// TwinCAT 3 PLC project PLC1
// ProgramVersion: 3.1.4024.0
// libraries:
//   Tc2_EtherCAT, * (Beckhoff Automation GmbH)
//   Tc2_Standard, * (Beckhoff Automation GmbH)
//   Tc2_System, * (Beckhoff Automation GmbH)
//   Tc2_Utilities, * (Beckhoff Automation GmbH)
//   Tc3_BA2_Common, * (Beckhoff Automation GmbH)
//   Tc3_Module, * (Beckhoff Automation GmbH)
// project tree:
//   DUTs/SMPTE Timecode/ E_SMPTE_AnalogValue.TcDUT, E_SMPTE_FrameMode.TcDUT, E_SMPTE_PartOfFrame.TcDUT, E_SMPTE_TimeController_Mode.TcDUT, E_SMPTE_TimeController_Source.TcDUT, ST_SMPTE_TimeStruct.TcDUT, ST_SMPTE_TimeStructExt.TcDUT
//   DUTs/ ST_EL4732_State.TcDUT
//   FBs/ FB_SMPTE_Receiver.TcPOU, FB_SMPTE_Sender.TcPOU, FB_SMPTE_TimeController.TcPOU
//   ITFs/ I_SMPTE_TimeController.TcIO
//   POUs/ MAIN_Sender.TcPOU, MAIN_Receiver.TcPOU
//   Tasks/ PlcTaskReceiver.TcTTO, PlcTaskSender.TcTTO
// real-time tasks:
//   TASK PlcTaskReceiver: cycle T#1ms, priority 20, ADS port 350
//   TASK PlcTaskSender: cycle T#20ms, priority 1, ADS port 351
// I/O:
//   DEVICE Device 7 (EtherCAT), AmsNetId 169.254.250.244.8.1
//     Term 1 (EK1100) [EK1100 EtherCAT Coupler (2A E-Bus)]
//       Term 2 (EL4732) [EL4732 2Ch. Ana. Output +/-10V, Oversample]
//       Term 3 (EL3702) [EL3702 2Ch. Ana. Input +/-10V, DIFF, Oversample]
//       Term 4 (EL9011) [EL9011 End Terminal]
// variable links:
//   PLC1/PLC1 Instance <-> Device 7 (EtherCAT)/Term 1 (EK1100)/Term 2 (EL4732)
//     PlcTaskSender Outputs/MAIN_Sender.SMPTE_Sender.aSMPTE_out[{0..79}] <-> Ch1 Sample {0..79}/Ch1 Value  (80 links)
//   PLC1/PLC1 Instance <-> Device 7 (EtherCAT)/Term 1 (EK1100)/Term 3 (EL3702)
//     PlcTaskReceiver Inputs/MAIN_Receiver.SMPTE_Receiver.EL3702_Samples[{1..100}] <-> Ch1 Sample {0..99}/Ch1 Value  (100 links)
//   PLC1/PLC1 Instance <-> TcCOM Objects/Object1 (TcDcExternalTimeProvider)
//     PlcTaskSender Inputs/MAIN_Sender.nSysTime <-> Outputs/nSysTime

CONFIGURATION PLC1
    RESOURCE PLC ON TwinCAT3
        TASK PlcTaskReceiver(INTERVAL := T#1ms, PRIORITY := 20);
        TASK PlcTaskSender(INTERVAL := T#20ms, PRIORITY := 1);
        PROGRAM MAIN_Receiver WITH PlcTaskReceiver : MAIN_Receiver;
        PROGRAM MAIN_Sender WITH PlcTaskSender : MAIN_Sender;
    END_RESOURCE
END_CONFIGURATION

// ---- DUTs/SMPTE Timecode/E_SMPTE_AnalogValue.TcDUT
TYPE E_SMPTE_AnalogValue :
(
	LOW := 0, HIGH := 32000
)INT;
END_TYPE

// ---- DUTs/SMPTE Timecode/E_SMPTE_FrameMode.TcDUT
{attribute 'qualified_only'}
{attribute 'strict'}
TYPE E_SMPTE_FrameMode :
(
	FPS_25
);
END_TYPE

// ---- DUTs/SMPTE Timecode/E_SMPTE_PartOfFrame.TcDUT
{attribute 'qualified_only'}
{attribute 'strict'}
TYPE E_SMPTE_PartOfFrame :
(
	first := 0, second := 1
)BYTE;
END_TYPE

// ---- DUTs/SMPTE Timecode/E_SMPTE_TimeController_Mode.TcDUT
{attribute 'qualified_only'}
{attribute 'strict'}
TYPE E_SMPTE_TimeController_Mode :
(
	Stopped := 0,
	Playing := 1,
	Paused := 2
);
END_TYPE

// ---- DUTs/SMPTE Timecode/E_SMPTE_TimeController_Source.TcDUT
{attribute 'qualified_only'}
{attribute 'strict'}
TYPE E_SMPTE_TimeController_Source :
(
	NT_Time := 0,
	DC_Time := 1,
	ExtTimeProvider := 2
);
END_TYPE

// ---- DUTs/SMPTE Timecode/ST_SMPTE_TimeStruct.TcDUT
TYPE ST_SMPTE_TimeStruct :
STRUCT
	Hours: BYTE; 		// 0..24 h
	Minutes: BYTE; 		// 0..60 min
	Seconds: BYTE;		// 0..60 sec
	Frames: BYTE;		// 0..24|25|30 frames
END_STRUCT
END_TYPE

// ---- DUTs/SMPTE Timecode/ST_SMPTE_TimeStructExt.TcDUT
// Extended time struct
TYPE ST_SMPTE_TimeStructExt EXTENDS ST_SMPTE_TimeStruct :
STRUCT
	FramesUnits: BYTE;
	FramesTens: BYTE;
	SecondsUnits: BYTE;
	SecondsTens: BYTE;
	MinutesUnits: BYTE;
	MinutesTens: BYTE;
	HoursUnits: BYTE;
	HoursTens: BYTE;
END_STRUCT
END_TYPE

// ---- DUTs/ST_EL4732_State.TcDUT
TYPE ST_EL4732_State :
STRUCT
	WcState AT %I*: BYTE;
	ImfoData_State AT %I*: UINT;
	InfoData_DcOutputShift AT %I*: DINT;
	InfoData_DDcInputShift AT %I*: DINT;
END_STRUCT
END_TYPE

// ---- ITFs/I_SMPTE_TimeController.TcIO
INTERFACE I_SMPTE_TimeController

METHOD Cycle : BOOL
VAR_INPUT
END_VAR
END_METHOD

// Will pause the time
METHOD Pause : BOOL
VAR_INPUT
	bExecute : BOOL;
END_VAR
END_METHOD

PROPERTY Paused : BOOL
GET
END_GET
END_PROPERTY

// Starts the time
METHOD Play : BOOL
VAR_INPUT
	bExecute : BOOL;
END_VAR
END_METHOD

PROPERTY Playing : BOOL
GET
END_GET
END_PROPERTY

// Resets the time
METHOD Reset : BOOL
VAR_INPUT
	bExecute : BOOL;
END_VAR
END_METHOD

// Will stop the time and reset to 00:00:00:00
METHOD Stop : BOOL
VAR_INPUT
	bExecute : BOOL;
END_VAR
END_METHOD

PROPERTY Stopped : BOOL
GET
END_GET
END_PROPERTY

// Returns the SMPTE_Sender_TimeStruct
PROPERTY TimeStruct : REFERENCE TO ST_SMPTE_TimeStruct;
GET
END_GET
END_PROPERTY

END_INTERFACE

// ---- POUs/MAIN_Receiver.TcPOU
PROGRAM MAIN_Receiver
VAR
	// SMPTE Receiver
	SMPTE_Receiver 	: FB_SMPTE_Receiver;
	ReceivingSignal	: BOOL;
	FrameRate		: REAL;
	TimeString		: STRING;
	TimeStruct		: ST_SMPTE_TimeStruct;
END_VAR

(************************)
(**** SMPTE Receiver ****)
(************************)

// Call the execute method once each cycle
SMPTE_Receiver.Cycle();
// Check if the cable is connected and receiving timecode analog signal
ReceivingSignal := SMPTE_Receiver.Receiving;
// Get the framerate
FrameRate := SMPTE_Receiver.FrameRate;
// Get the time as string output
TimeString := SMPTE_Receiver.TimeString;
// Get the time as time struct
TimeStruct := SMPTE_Receiver.TimeStruct;

END_PROGRAM

// ---- FBs/FB_SMPTE_Receiver.TcPOU
FUNCTION_BLOCK FB_SMPTE_Receiver
VAR
	EL3702_Samples AT %I*: ARRAY[1..OversamplingFactor] OF INT;
	EL3702_Samples_Doublecycles : ARRAY[1..DoubleOversamplingFactor] OF INT;
	EL3702_Samples_DoublecyclesTrig : ARRAY[1..DoubleOversamplingFactor] OF INT;
	Tab_TimeCodeFrame: ARRAY[1..TimeCodeFrame] OF BYTE;					(* Bit read in the frame *)
	LastTimeCodeFrame: ARRAY[0..79] OF BYTE;									(* Last and unique TimeCode Frame *)
	SyncWord : ARRAY [1..16] OF BYTE :=[ 0, 0, 1, 1, 1, 1, 1, 1, 1, 1, 1, 1, 1, 1, 0, 1];
	SyncWordTemp : ARRAY [1..16] OF BYTE;
	i: WORD;
	j: DWORD;
	LastEdge: DWORD;
	ConstantTime: DWORD;
	Even: BOOL;	(* Is use to mesure 2 half period to detect a bit 1 *)
	First_BitZero_Reach: BOOL  := FALSE ;	(* We can mesure only when we reach a first Bit 0 otherwise we do not know in which half period of a bit 1 we are *)
	Index_Tab_EL3702: INT := 102;
	Index_Tab_TimeCodeFrame: WORD := 1;
	h: WORD;

	Index_Tab_EL3702_Error: WORD;			(* Increased when an edge had not beed detected in the last cycle *)
	Index_Tab_TimeCodeFrame_Error: WORD;	(* Increased when we are not able to catch a SyncWord in the big Array of TimeCode Bits. Normally, an Syncword each 80 bits *)
	
	// Internal Properties
	_Reset : BOOL;
	_Receiving : BOOL;
	_FrameRate: REAL;
	_FrameError: DWORD;
	
	_SMPTE_TimeStruct : ST_SMPTE_TimeStruct;
	_SMPTE_TimeStructExt : ST_SMPTE_TimeStructExt;

	_FrameRead: DWORD;
	_Time_String: STRING;
END_VAR

VAR CONSTANT
	OversamplingFactor: WORD := 100;			(* EL3702 Oversampling rate = 100 samples per cycle *)
	DoubleOversamplingFactor: WORD := 200;	(*  = OversamplingFactor x 2 *)
	TimeCodeFrame : WORD := 300;				(* bits detected in the Timecode signal *)
	SignalThreshold : INT := 25;
END_VAR

METHOD Cycle : BOOL
VAR_INST
	// Check if there is a timing error
	rtTimeError : R_TRIG;
END_VAR
// Check timing error and task time
rtTimeError(CLK := UDINT_TO_LREAL(_TaskInfo[GETCURTASKINDEXEX()].CycleTime) / 10_000 <> 1);
IF rtTimeError.Q THEN
	ADSLOGSTR( msgCtrlMask := ADSLOG_MSGTYPE_ERROR OR ADSLOG_MSGTYPE_MSGBOX, msgFmtStr := 'PLC SMPTE Receiver: Execution Time Not Valid, Please set to 1ms','');
END_IF

IF _Reset THEN
	First_BitZero_Reach := FALSE;
	Index_Tab_TimeCodeFrame := 1;
	Index_Tab_EL3702 := 102;
	Even := FALSE;
	FOR i:= 1 TO TimeCodeFrame DO
		Tab_TimeCodeFrame [ i ] := 0;
	END_FOR
	_Reset := FALSE;
END_IF

IF SignalCheck() THEN
	(* We save the last 2 cycles *)
	FOR i:=1 TO OversamplingFactor DO
		EL3702_Samples_Doublecycles [ i ] := EL3702_Samples_Doublecycles [ i+OversamplingFactor ];
	END_FOR
	FOR i:=1 TO OversamplingFactor DO
		EL3702_Samples_Doublecycles [ OversamplingFactor + i ] := EL3702_Samples [i];
	END_FOR
	
	(* Now we create an ARRAY that show the binary code *)
	ConstantTime := 0;							(* ConstantTime is the duration of a constant level of the analog signal, time between 2 edges *)
	FOR i:= 1 TO 2*OversamplingFactor DO
		  EL3702_Samples_DoublecyclesTrig [i ] := 0;	(* An array that provide only the edges of the analog signal, only in the last cycle *)
	END_FOR
	
	FOR i:= Index_Tab_EL3702 TO ( 2*OversamplingFactor-1)  DO
		IF 	EL3702_Samples_Doublecycles[ i-1] * EL3702_Samples_Doublecycles [ i ] < 0					(* The analog signal change of sign --> there is an edge *)
		OR 	EL3702_Samples_Doublecycles [ i-1 ] <> 0 AND EL3702_Samples_Doublecycles [ i ] = 0 THEN	(* We capture a sample that is 0 : It's also a new edge *)
			EL3702_Samples_DoublecyclesTrig [ i ] := 1;
			IF LastEdge = 0 THEN										(* We have to wait a least the second edge to mesure *)
				LastEdge := i;
			ELSE													(* Let's go ... *)
				ConstantTime := (i - LastEdge) * 10 ;  	(* if  EL3702 Oversampling time = 10 µs*)
				LastEdge := i;
				IF ConstantTime < 330 AND ConstantTime<>0 AND First_BitZero_Reach THEN		(* It's part of a 1 signal *)
					(* 330µs is a fix limit that match all frame rates : Minimum period is 400 µs at 30 fr/sec, maximum half period is 260 µs at 24 fr/sec*)
					IF First_BitZero_Reach THEN											(* We first need to read a 0 bit, or we are not able to know in wich part of a 1 bit we are *)
						IF NOT Even THEN				(* First part of a 1 bit *)
							Index_Tab_EL3702 := i ;
							Even := TRUE;
						ELSE							(* Second part of a 1 bit *)
							Tab_TimeCodeFrame [ Index_Tab_TimeCodeFrame ] := 1;			(* We save a 1 bit in an array *)
							Index_Tab_TimeCodeFrame := Index_Tab_TimeCodeFrame + 1;		(* and manage this array *)
							Index_Tab_EL3702 := i ;										(* This bit in Frame is already handled, we will continu from this sample *)
							Even := FALSE;
						END_IF
					END_IF
				ELSIF ConstantTime > 300  THEN											(* It's a 0 bit *)
					First_BitZero_Reach := TRUE; 											(* One 0 bit had been detected. We are now able to mesure 1 bit *)
					IF Even THEN						(* If we were in the first part of a 1 bit *)
						Even := FALSE;
						_FrameError := _FrameError + 1;		(* Then this 1 bit is not finished and it's a Frame Error *)
					END_IF
					Tab_TimeCodeFrame [ Index_Tab_TimeCodeFrame ] := 0;					(* We save a 1 bit in an array *)
					Index_Tab_TimeCodeFrame := Index_Tab_TimeCodeFrame + 1;				(* and manage this array *)
					Index_Tab_EL3702 := i ;												(* This bit in Frame is already handled, we will continu from this sample *)
					_FrameRate := 1000000.0 / (ConstantTime * 80);	(* We measure the frame Rate. 0 Signal = 1 bit. 80 bit / frame *)
				END_IF
			END_IF
		END_IF
	END_FOR
	Index_Tab_EL3702 := Index_Tab_EL3702 - OversamplingFactor +1; 			(* +1 in order to do not take in consideration the last one we handled *)
	IF Index_Tab_EL3702 < 2  THEN							(* There is a problem : We should be able to read an edge in the last cycle *)
		Index_Tab_EL3702_Error := Index_Tab_EL3702_Error + 1;
	END_IF
	LastEdge := LastEdge - OversamplingFactor;										(* We will shift the array of the last 2 Oversampling cycle. Then the last Edge will be 100 samples before *)
	
	
	
	
	(* We are looking for the SyncWord - Sequence 0, 0, 1, 1, 1, 1, 1, 1, 1, 1, 1, 1, 1, 1, 0, 1 *)
	FOR i:=16 TO  ( TimeCodeFrame ) DO	(* Sync Word = 16 bits *)
		FOR j := 1 TO 16 DO
			SyncWordTemp [ j ] := Tab_TimeCodeFrame [ i -16 + j ]; 				(* Part of the Array that contain all bits read from the Timecode Frame *)
		END_FOR
		IF MEMCMP( ADR(SyncWord) , ADR(SyncWordTemp), 16) = 0 THEN		(* We compare this part with the SynWord *)
			IF i >= 80 THEN	(* A SyncWord is found and all bits that are in this frame are available *)
					MEMCPY( ADR(LastTimeCodeFrame) , ADR(Tab_TimeCodeFrame) + i  - 80, 80);	(* We extract this TimeCode Frame from the complete array *)
					
					_SMPTE_TimeStructExt.FramesUnits := LastTimeCodeFrame [0] * 1
													+LastTimeCodeFrame [1] * 2
													+LastTimeCodeFrame [2] * 4
													+LastTimeCodeFrame [3] * 8;
													
					_SMPTE_TimeStructExt.FramesTens :=  LastTimeCodeFrame [8] * 10
													+LastTimeCodeFrame [9] * 20;
													
					_SMPTE_TimeStructExt.SecondsUnits := LastTimeCodeFrame [16] * 1
													 +LastTimeCodeFrame [17] * 2
													 +LastTimeCodeFrame [18] * 4
													 +LastTimeCodeFrame [19] * 8;
													 
					_SMPTE_TimeStructExt.SecondsTens := LastTimeCodeFrame [24] * 10
													+LastTimeCodeFrame [25] * 20
													+LastTimeCodeFrame [26] * 40;
													
					_SMPTE_TimeStructExt.MinutesUnits := LastTimeCodeFrame [32] * 1
													 +LastTimeCodeFrame [33] * 2
													 +LastTimeCodeFrame [34] * 4
													 +LastTimeCodeFrame [35] * 8;
													 
					_SMPTE_TimeStructExt.MinutesTens := LastTimeCodeFrame [40] * 10
													+LastTimeCodeFrame [41] * 20
													+LastTimeCodeFrame [42] * 40;
													
					_SMPTE_TimeStructExt.HoursUnits := LastTimeCodeFrame [48] * 1
												   +LastTimeCodeFrame [49] * 2
												   +LastTimeCodeFrame [50] * 4
												   +LastTimeCodeFrame [51] * 8;
												   
					_SMPTE_TimeStructExt.HoursTens := LastTimeCodeFrame [56] * 10
												   +LastTimeCodeFrame [57] * 20;
												   

					_SMPTE_TimeStructExt.Frames := _SMPTE_TimeStructExt.FramesTens + _SMPTE_TimeStructExt.FramesUnits;
					_SMPTE_TimeStructExt.Seconds := _SMPTE_TimeStructExt.SecondsTens + _SMPTE_TimeStructExt.SecondsUnits;
					_SMPTE_TimeStructExt.Minutes := _SMPTE_TimeStructExt.MinutesTens + _SMPTE_TimeStructExt.MinutesUnits;
					_SMPTE_TimeStructExt.Hours := _SMPTE_TimeStructExt.HoursTens + _SMPTE_TimeStructExt.HoursUnits;
					
					_SMPTE_TimeStruct.Frames  := _SMPTE_TimeStructExt.Frames;
					_SMPTE_TimeStruct.Seconds := _SMPTE_TimeStructExt.Seconds;
					_SMPTE_TimeStruct.Minutes := _SMPTE_TimeStructExt.Minutes;
					_SMPTE_TimeStruct.Hours   := _SMPTE_TimeStructExt.Hours;
					
					_Time_String := CONCAT ( INT_TO_STRING (_SMPTE_TimeStructExt.Hours), ' : ');
					_Time_String := CONCAT (_Time_String,  INT_TO_STRING (_SMPTE_TimeStructExt.Minutes));
					_Time_String := CONCAT (_Time_String,  ' : ');
					_Time_String := CONCAT (_Time_String,  INT_TO_STRING (_SMPTE_TimeStructExt.Seconds));
					_Time_String := CONCAT (_Time_String,  ' : ');
					_Time_String := CONCAT (_Time_String,  INT_TO_STRING (_SMPTE_TimeStructExt.Frames));
	
					_FrameRead := _FrameRead + 1; 							(* Number of frame read *)
	
					FOR h:=1 TO (TimeCodeFrame - i ) DO							(* Now, we suppress this TimeCode frame from the array of bit, and shift this array *)
						Tab_TimeCodeFrame [ h ] := Tab_TimeCodeFrame [ h + i ];
					END_FOR
					FOR h:= (TimeCodeFrame - i ) TO TimeCodeFrame DO
						Tab_TimeCodeFrame [ h ] := 0;
					END_FOR
	
					 Index_Tab_TimeCodeFrame := Index_Tab_TimeCodeFrame - i ;		(* Next bit in the frame will be place here now *)
	
					EXIT ;
			END_IF
		END_IF
	END_FOR
	
	IF Index_Tab_TimeCodeFrame > TimeCodeFrame THEN	(* There is a problem : We should be able to catch a SyncWord in a so big array a Timecode bit. Normally a SyncWord each 80 bits*)
		Index_Tab_TimeCodeFrame_Error := Index_Tab_TimeCodeFrame_Error + 1;
		Reset := TRUE;
	END_IF
END_IF
END_METHOD

PROPERTY FrameError : DWORD
GET
FrameError := _FrameError;
END_GET
END_PROPERTY

PROPERTY FrameRate : REAL
GET
FrameRate := _FrameRate;
END_GET
END_PROPERTY

PROPERTY FramesReceived : DWORD
GET
FramesReceived := _FrameRead;
END_GET
END_PROPERTY

PROPERTY Receiving : BOOL
GET
Receiving := _Receiving;
END_GET
END_PROPERTY

PROPERTY Reset : BOOL
SET
_Reset := Reset;
END_SET
END_PROPERTY

METHOD INTERNAL SignalCheck : BOOL
VAR
	itr_X : INT;
END_VAR
// Check for EL3702 is receiving signals, plugged into device
_Receiving := FALSE;
FOR itr_X := 1 TO 100 DO
	IF EL3702_Samples[itr_X] >= SignalThreshold OR EL3702_Samples[itr_X] <= (SignalThreshold * -1) THEN
		SignalCheck := TRUE;
		_Receiving := TRUE;
		EXIT;
	END_IF
END_FOR
END_METHOD

PROPERTY TimeString : REFERENCE TO STRING
GET
TimeString REF= _Time_String;
END_GET
END_PROPERTY

PROPERTY TimeStruct : REFERENCE TO ST_SMPTE_TimeStruct
GET
TimeStruct REF= _SMPTE_TimeStruct;
END_GET
END_PROPERTY

PROPERTY TimeStructExt : REFERENCE TO ST_SMPTE_TimeStructExt
GET
TimeStructExt REF= _SMPTE_TimeStructExt;
END_GET
END_PROPERTY

END_FUNCTION_BLOCK

// ---- POUs/MAIN_Sender.TcPOU
PROGRAM MAIN_Sender
VAR
	// SMPTE Time Controller
	SMPTE_TimeController : FB_SMPTE_TimeController(eTimeSource := E_SMPTE_TimeController_Source.ExtTimeProvider, eFrameMode := E_SMPTE_FrameMode.FPS_25);
	// SMPTE Sender
	SMPTE_Sender 	: FB_SMPTE_Sender(ipSMPTE_TimeController := SMPTE_TimeController);
	
	// External Time Source
	nSysTime AT %I* : ULINT;
	
	// Enable the sender
	bEnableSending: BOOL;
	// Disable the sender
	bDisableSending: BOOL;
	// Error status of sender
	bSMPTE_Error: BOOL;
	// Enable Status
	bSMPTE_Enabled: BOOL;
	
	// Play the timeline
	bPlay: BOOL;
	// Pause the timeline
	bPause: BOOL;
	// Stop the timeline
	bStop: BOOL;
	// Reset the timeline
	bReset: BOOL;
	
	// View the current time struct being send
	stSMPTE_TimeStruct : ST_SMPTE_TimeStruct;

END_VAR

(**********************)
(**** SMPTE Sender ****)
(**********************)

// Call once each cycle
SMPTE_TimeController.Cycle();
SMPTE_Sender.Cycle();

// Enable sending the SMPTE signal
IF SMPTE_Sender.EnableSending(bExecute := bEnableSending) THEN
	bEnableSending := FALSE;
END_IF

// Disable sending the SMPTE signal
IF SMPTE_Sender.DisableSending(bExecute := bDisableSending) THEN
	bDisableSending := FALSE;
END_IF

// Check if errors on SMPTE Sender
bSMPTE_Error := SMPTE_Sender.Error;
// Check if enabled
bSMPTE_Enabled := SMPTE_Sender.Enabled;



(********************************)
(**** SMPTE Time Conectoller ****)
(********************************)

// Assign External Time Source
SMPTE_TimeController.AssignExternalTimeSource(nSysTime);

// Playback controls
IF SMPTE_TimeController.Play(bExecute := bPlay) THEN
	bPlay := FALSE;
END_IF

IF SMPTE_TimeController.Pause(bExecute := bPause) THEN
	bPause := FALSE;
END_IF

IF SMPTE_TimeController.Stop(bExecute := bStop) THEN
	bStop := FALSE;
END_IF

IF SMPTE_TimeController.Reset(bExecute := bReset) THEN
	bReset := FALSE;
END_IF

// Sample of Timecode being send
stSMPTE_TimeStruct := SMPTE_TimeController.TimeStruct;

END_PROGRAM

// ---- FBs/FB_SMPTE_TimeController.TcPOU
FUNCTION_BLOCK FB_SMPTE_TimeController IMPLEMENTS I_SMPTE_TimeController
VAR
	// Internal Time Source mode
	_eTimeSource : E_SMPTE_TimeController_Source;
	
	// Linked to TcCom Object for Time Provider if using Ext Mode
	_TcExternalTimeSource : REFERENCE TO ULINT; 
	
	// Frame Mode
	_eFrameMode: E_SMPTE_FrameMode := E_SMPTE_FrameMode.FPS_25;	// transmitting with 25 fps (frames per second)		
	
	// Used for DC Time
	_dcTime	: T_DCTIME64;
			
	// SMPTE Time Struct
	_stSMPTE_TimeStruct : ST_SMPTE_TimeStruct;
	
	// Reference time timestamp
	_bRefTimeInit : BOOL;
	
	// Current Time Strunct
	_CurrentTime :	TIMESTRUCT;
		
	// Current Time Value
	_RefTime : T_DCTIME64;
	
	// Working Time Value
	_WorkTime : T_DCTIME64;
	
	// Paused Time Value
	_PauseTime : T_DCTIME64;
	
	// Mode Status
	_eSMPTE_TimeController_Mode : E_SMPTE_TimeController_Mode;
	
	// Playing Status Variables
	_Playing : BOOL;
	
	// Paused Status Variables
	_Paused : BOOL;
	
	// Stopped Status Variables
	_Stopped : BOOL;
	
	// Reset Control Variables
	_Reset : BOOL;
	
	// Error, usually due to timesource
	_Error : BOOL;
END_VAR

METHOD AssignExternalTimeSource : BOOL
VAR_INPUT
	// Linked to TcCom Object for Time Provider if using Ext Mode
	TcExternalTimeSource : REFERENCE TO ULINT; 
END_VAR
_TcExternalTimeSource REF= TcExternalTimeSource;
AssignExternalTimeSource := TRUE;
END_METHOD

METHOD Cycle : BOOL
VAR_INST
	_CalcTimeDiff : FB_EcExtSyncCalcTimeDiff64;
	_bWasPaused : BOOL;
END_VAR
// Check Mode and compute time
CASE _eSMPTE_TimeController_Mode OF
	E_SMPTE_TimeController_Mode.Playing:
	
		// Get the working time
		UpdateTime(_WorkTime); 
		
		// Get the reference clock
		IF NOT _bRefTimeInit THEN
			_RefTime := _WorkTime;
			_bRefTimeInit := TRUE;
		END_IF
		
		// Recovery from Pause
		IF _bWasPaused THEN
			_RefTime := _WorkTime - _PauseTime;
			_bWasPaused := FALSE;
		END_IF

	E_SMPTE_TimeController_Mode.Paused:
		IF NOT _bWasPaused THEN
			_PauseTime := _WorkTime - _RefTime;
			_bWasPaused := TRUE;
		END_IF
	
	E_SMPTE_TimeController_Mode.Stopped:
		// Stop the clock and reset
		_bRefTimeInit := FALSE;
		_bWasPaused := FALSE;
		_PauseTime := 0;
		_WorkTime := 0;
		_RefTime := 0;
END_CASE

// If not paused, update the time stuct
IF NOT (_eSMPTE_TimeController_Mode = E_SMPTE_TimeController_Mode.Paused) THEN
	// Convert to time struct
	_CurrentTime := DCTIME64_TO_SYSTEMTIME(_WorkTime - _RefTime);
END_IF

// Reset
IF _Reset THEN
	_bRefTimeInit := FALSE;
	_bWasPaused := FALSE;
	_PauseTime := 0;
	_WorkTime := 0;
	_RefTime := 0;
	_Reset := FALSE;
END_IF

// Remove unused values
_CurrentTime.wDay := 0;
_CurrentTime.wDayOfWeek := 0;
_CurrentTime.wMonth := 0;
_CurrentTime.wYear := 0;
END_METHOD

PROPERTY Error : BOOL
GET
Error := _Error;
END_GET
END_PROPERTY

METHOD FB_init : BOOL
VAR_INPUT
	(* if TRUE, the retain variables are initialized (warm start / cold start)*)
	bInitRetains	: BOOL;
	(* if TRUE, the instance afterwards gets moved into the copy code (online change)*)
	bInCopyCode	: BOOL;
	(* Time Source*)
	eTimeSource	: E_SMPTE_TimeController_Source;
	(* Frame Mode, transmitting with 25 fps (frames per second) *)
	eFrameMode : E_SMPTE_FrameMode := E_SMPTE_FrameMode.FPS_25;
END_VAR
_eTimeSource := eTimeSource;
_eFrameMode := eFrameMode;
END_METHOD

(* Will pause the time*)
METHOD Pause : BOOL
VAR_INPUT
	bExecute	: BOOL;
END_VAR
VAR_INST
	rtExecute : R_TRIG;
END_VAR
rtExecute(CLK := bExecute);
IF rtExecute.Q THEN
	_eSMPTE_TimeController_Mode := E_SMPTE_TimeController_Mode.Paused;
	// Return TRUE
	Pause := TRUE;
END_IF
END_METHOD

PROPERTY Paused : BOOL
GET
Paused := _eSMPTE_TimeController_Mode = E_SMPTE_TimeController_Mode.Paused;
END_GET
END_PROPERTY

(* Starts the time*)
METHOD Play : BOOL
VAR_INPUT
	bExecute	: BOOL;
END_VAR
VAR_INST
	rtExecute :  R_TRIG;
END_VAR
rtExecute(CLK := bExecute);
IF rtExecute.Q THEN
	_eSMPTE_TimeController_Mode := E_SMPTE_TimeController_Mode.Playing;
	// Return TRUE
	Play := TRUE;
END_IF
END_METHOD

PROPERTY Playing : BOOL
GET
Playing := _eSMPTE_TimeController_Mode = E_SMPTE_TimeController_Mode.Playing;
END_GET
END_PROPERTY

(* Resets the time*)
METHOD Reset : BOOL
VAR_INPUT
	bExecute	: BOOL;
END_VAR
VAR_INST
	rtExecute :  R_TRIG;
END_VAR
rtExecute(CLK := bExecute);
IF rtExecute.Q THEN
	_Reset := TRUE;
	// Return TRUE
	Reset := TRUE;
END_IF
END_METHOD

(* Will stop the time and reset to 00:00:00:00*)
METHOD Stop : BOOL
VAR_INPUT
	bExecute	: BOOL;
END_VAR
VAR_INST
	rtExecute :  R_TRIG;
END_VAR
rtExecute(CLK := bExecute);
IF rtExecute.Q THEN
	_eSMPTE_TimeController_Mode := E_SMPTE_TimeController_Mode.Stopped;
	// Return TRUE
	Stop := TRUE;
END_IF
END_METHOD

PROPERTY Stopped : BOOL
GET
Stopped := _eSMPTE_TimeController_Mode = E_SMPTE_TimeController_Mode.Stopped;
END_GET
END_PROPERTY

(* Returns the SMPTE_TimeStruct*)
PROPERTY TimeStruct : REFERENCE TO ST_SMPTE_TimeStruct;
GET
// Compute the Time Struct for SMPTE
CASE _eFrameMode OF
	E_SMPTE_FrameMode.FPS_25:
		_stSMPTE_TimeStruct.Hours := WORD_TO_BYTE(_CurrentTime.wHour);
		_stSMPTE_TimeStruct.Minutes := WORD_TO_BYTE(_CurrentTime.wMinute);
		_stSMPTE_TimeStruct.Seconds := WORD_TO_BYTE(_CurrentTime.wSecond);
		_stSMPTE_TimeStruct.Frames := DINT_TO_BYTE(TRUNC(WORD_TO_REAL(_CurrentTime.wMilliseconds)/(1000/25)));
END_CASE

// Return the time struct
TimeStruct REF= _stSMPTE_TimeStruct;
END_GET
END_PROPERTY

METHOD INTERNAL UpdateTime: BOOL;
VAR_IN_OUT
	// Current Time Struct
	_CurDCTime : T_DCTIME64;
END_VAR
VAR_INST
	// Used for NT Time
	_ntTime	: TIMESTRUCT;
	_ntGetTime : NT_GetTime;
	// Ref Error Trig
	rtRefError : R_TRIG; 
END_VAR
// Check for reference error on External time source
rtRefError(CLK := NOT __ISVALIDREF(_TcExternalTimeSource));
IF rtRefError.Q THEN
	ADSLOGSTR( msgCtrlMask := ADSLOG_MSGTYPE_ERROR OR ADSLOG_MSGTYPE_MSGBOX, msgFmtStr := 'PLC SMPTE Time Controller: Invalid Timesource Provided or Disconnected: Use AssignExternalTimeSource()','');
END_IF

// Calculate the time
CASE _eTimeSource OF
	E_SMPTE_TimeController_Source.ExtTimeProvider:
		(* External Time Provider *)
		IF __ISVALIDREF(_TcExternalTimeSource) THEN
			_dcTime := FILETIME64_TO_DCTIME64(_TcExternalTimeSource);
			_CurDCTime := _dcTime;
			_Error := FALSE;
		ELSE
			_eSMPTE_TimeController_Mode := E_SMPTE_TimeController_Mode.Stopped;
			_Error := TRUE;
		END_IF
	
	E_SMPTE_TimeController_Source.DC_Time:
		(* External Time Provider *)
		_dcTime := F_GetCurDcTickTime64();
		_CurDCTime := _dcTime;
	
	E_SMPTE_TimeController_Source.NT_Time:
		(* NT Time Provider *)
		IF NOT _ntGetTime.BUSY THEN
			_ntGetTime(start := TRUE, TIMESTR => _ntTime);
		END_IF
		_ntGetTime(start := FALSE);
		_CurDCTime := SYSTEMTIME_TO_DCTIME64(_ntTime, 0, 0);
END_CASE

UpdateTime := TRUE;
END_METHOD

END_FUNCTION_BLOCK

// ---- FBs/FB_SMPTE_Sender.TcPOU
FUNCTION_BLOCK FB_SMPTE_Sender
VAR
	// Analog Signal Output
	aSMPTE_out AT%Q*: ARRAY[0..79] OF E_SMPTE_AnalogValue;
	
	// Status Variables
	_bEnabled: BOOL; // Enabled
	_bError: BOOL;	// becomes true, if plc cycle time <> 20ms	
	_bReady: BOOL;	// two cycles are needed to transmitt a comlete message - the FB accepts data only if READY!
	
	// SMPTE Time Contrller Object
	_ipSMPTE_TimeController : I_SMPTE_TimeController;
		
	// Internal Variables
	eCurrentPart: E_SMPTE_PartOfFrame := E_SMPTE_PartOfFrame.first;
	nPos: BYTE;
	aTmp: ARRAY[0..3] OF BOOL;

	// Internal Time Struct
	_stSMPTE_TimeStruct: ST_SMPTE_TimeStruct;
END_VAR

METHOD INTERNAL ChangePart  : HResult
VAR_IN_OUT
	eCurrentPartOfFrame : E_SMPTE_PartOfFrame;
END_VAR
eCurrentPartOfFrame := sel(eCurrentPartOfFrame = E_SMPTE_PartOfFrame.first, E_SMPTE_PartOfFrame.first, E_SMPTE_PartOfFrame.second);
END_METHOD

METHOD Cycle : BOOL
VAR_INST
	rTrigEnable: R_TRIG;
	fTrigEnable: F_TRIG;
	// Check if there is a timing error
	rtTimeError : R_TRIG;
END_VAR
// Check timing error and task time
rtTimeError(CLK := UDINT_TO_LREAL(_TaskInfo[GETCURTASKINDEXEX()].CycleTime) / 10_000 <> 20);
IF rtTimeError.Q THEN
	ADSLOGSTR( msgCtrlMask := ADSLOG_MSGTYPE_ERROR OR ADSLOG_MSGTYPE_MSGBOX, msgFmtStr := 'PLC SMPTE Sender: Execution Time Not Valid, Please set to 20ms','');
END_IF

rTrigEnable(CLK := _bEnabled);
fTrigEnable(CLK := _bEnabled);

IF fTrigEnable.Q THEN
	_bReady := FALSE;
ELSIF rTrigEnable.Q THEN
	eCurrentPart := E_SMPTE_PartOfFrame.first;
	// cycle time using this FB must be 20ms - reason: Oversampling terminal!
	_bError := UDINT_TO_LREAL(_TaskInfo[GETCURTASKINDEXEX()].CycleTime) / 10_000 <> 20;
END_IF	

// Check if time source is valid and configured
IF (_ipSMPTE_TimeController = 0) THEN
	_bError := TRUE;
END_IF

// Check if there are errors or if no enabled
IF NOT _bEnabled OR _bError THEN
	RETURN;
END_IF
	
nPos := 0;
IF eCurrentPart = E_SMPTE_PartOfFrame.first THEN
	_stSMPTE_TimeStruct := _ipSMPTE_TimeController.TimeStruct;	// accept input value now!
	{region 'Frames (including userbits)'}
	Write_4Bits(aSMPTE_out,nPos, GetBits(_stSMPTE_TimeStruct.Frames, FALSE));
	Write_4Bits(aSMPTE_out,nPos, GetBits(0, TRUE));          
	Write_4Bits(aSMPTE_out,nPos, GetBits(_stSMPTE_TimeStruct.Frames,TRUE));
	Write_4Bits(aSMPTE_out,nPos, GetBits(0, TRUE));          
	{endregion}                                              
                                                             
	{region 'Seconds (including userbits'}                   
	Write_4Bits(aSMPTE_out,nPos, GetBits(_stSMPTE_TimeStruct.Seconds, FALSE));
	Write_4Bits(aSMPTE_out,nPos, GetBits(0, TRUE));          
	Write_4Bits(aSMPTE_out,nPos, GetBits(_stSMPTE_TimeStruct.Seconds,TRUE));
	Write_4Bits(aSMPTE_out,nPos, GetBits(0, TRUE));          
	{endregion}                                              
                                                             
	{region 'Minutes - Units only!'}                         
	Write_4Bits(aSMPTE_out,nPos, GetBits(_stSMPTE_TimeStruct.Minutes, FALSE));
	Write_4Bits(aSMPTE_out,nPos, GetBits(0, TRUE));          
	{endregion}                                              
                                                             
	_bReady := FALSE; 	                                     
		                                                     
ELSE // second part of the complete SMPTE Frame              
	{region 'Minutes - Tens only!'}                          
	Write_4Bits(aSMPTE_out,nPos, GetBits(_stSMPTE_TimeStruct.Minutes, TRUE));
	Write_4Bits(aSMPTE_out,nPos, GetBits(0, TRUE));          
	{endregion}                                              
                                                             
	{region 'hours (including userbits'}                     
	Write_4Bits(aSMPTE_out,nPos, GetBits(_stSMPTE_TimeStruct.Hours, FALSE));
	Write_4Bits(aSMPTE_out,nPos, GetBits(0, TRUE));          
	Write_4Bits(aSMPTE_out,nPos, GetBits(_stSMPTE_TimeStruct.Hours,TRUE));
	Write_4Bits(aSMPTE_out,nPos, GetBits(0, TRUE));
	{endregion}

	{region 'Syncword'}
	WriteSyncWord(aSMPTE_out,nPos);
	{endregion}
		 
	_bReady := TRUE;			 
END_IF

// one complete SMPTE frame always consists of two parts (2*20ms):
ChangePart(eCurrentPartOfFrame := eCurrentPart);
END_METHOD

METHOD DisableSending : BOOL
VAR_INPUT
	bExecute	: BOOL;
END_VAR
VAR_INST
	rtExecute : R_TRIG;
END_VAR
rtExecute(CLK := bExecute);
IF rtExecute.Q THEN
	_bEnabled := FALSE;
	// Return TRUE
	DisableSending := TRUE;
END_IF
END_METHOD

PROPERTY Enabled : BOOL
GET
Enabled := _bEnabled;
END_GET
END_PROPERTY

METHOD EnableSending : BOOL
VAR_INPUT
	bExecute	: BOOL;
END_VAR
VAR_INST
	rtExecute : R_TRIG;
END_VAR
rtExecute(CLK := bExecute);
IF rtExecute.Q THEN
	_bEnabled := TRUE;
	// Return TRUE
	EnableSending := TRUE;
END_IF
END_METHOD

PROPERTY Error : BOOL
GET
END_GET
END_PROPERTY

METHOD FB_init : BOOL
VAR_INPUT
	bInitRetains : BOOL; // if TRUE, the retain variables are initialized (warm start / cold start)
	bInCopyCode : BOOL;  // if TRUE, the instance afterwards gets moved into the copy code (online change)
	ipSMPTE_TimeController : I_SMPTE_TimeController;
END_VAR
_ipSMPTE_TimeController := ipSMPTE_TimeController;
END_METHOD

METHOD INTERNAL GetBits : ARRAY[0..3] OF BOOL
VAR_INPUT
	nValue: BYTE;
	bGetTens: BOOL;
END_VAR
VAR
	i: SINT;
END_VAR
FOR i:= 3 TO 0 BY -1 DO
	GetBits[i] := nValue >= 10* EXPT(2,i);
	nValue := LREAL_TO_BYTE(SEL(GetBits[i], nValue, nValue - (10* EXPT(2,i))));
END_FOR

IF bGetTens THEN
	RETURN;
END_IF

FOR i:= 3 TO 0 BY -1 DO
	GetBits[i] := nValue >= EXPT(2,i);
	nValue := LREAL_TO_BYTE(SEL(GetBits[i], nValue, nValue - EXPT(2,i)));
END_FOR
END_METHOD

PROPERTY Ready : BOOL
GET
END_GET
END_PROPERTY

METHOD INTERNAL Write_4Bits : HResult
VAR_IN_OUT
	aDataOut: ARRAY[0..79] OF E_SMPTE_AnalogValue;
	nPos: BYTE;
END_VAR

VAR_input
	aValue: ARRAY[0..3] OF BOOL;
END_VAR

VAR
	ePreviousAnalogValue: E_SMPTE_AnalogValue;
	i: SINT;
END_VAR
IF nPos = 0 THEN
	ePreviousAnalogValue := aDataOut[79];
	Write_4Bits := 1;
ELSE
	ePreviousAnalogValue := aDataOut[nPos-1];
	Write_4Bits := S_OK;
END_IF

FOR i:= 0 TO 3 DO
	IF aValue[i] THEN
		IF ePreviousAnalogValue = E_SMPTE_AnalogValue.HIGH THEN
			aDataOut[nPos] := E_SMPTE_AnalogValue.LOW;
			aDataOut[nPos + 1] := E_SMPTE_AnalogValue.HIGH;
		ELSE
			aDataOut[nPos] := E_SMPTE_AnalogValue.HIGH;
			aDataOut[nPos + 1] := E_SMPTE_AnalogValue.LOW;
		END_IF
	ELSE
		IF ePreviousAnalogValue = E_SMPTE_AnalogValue.HIGH THEN
			aDataOut[nPos] := aDataOut[nPos + 1] := E_SMPTE_AnalogValue.LOW;
		ELSE
			aDataOut[nPos] := aDataOut[nPos + 1] := E_SMPTE_AnalogValue.HIGH;
		END_IF
	END_IF
	ePreviousAnalogValue := aDataOut[nPos + 1];
	nPos := nPos + 2;
END_FOR
END_METHOD

METHOD INTERNAL WriteSyncword: HRESULT
VAR_IN_OUT
	aDataOut: ARRAY[0..79] OF E_SMPTE_AnalogValue;
	nPos: BYTE;
END_VAR

VAR
	i: INT;
END_VAR
// Syncword: 0011.1111.1111.1101

WriteSyncword	:= S_OK;
IF nPos <> 48 THEN
	WriteSyncword	:= -3;
	RETURN;
ELSIF aDataOut[47]=  E_SMPTE_AnalogValue.HIGH THEN // create syncword based on the last analog value ...
	// 0011
	aDataOut[nPos] := E_SMPTE_AnalogValue.LOW; 		nPos := nPos + 1;
	aDataOut[nPos] := E_SMPTE_AnalogValue.LOW; 		nPos := nPos + 1;
	aDataOut[nPos] := E_SMPTE_AnalogValue.HIGH; 		nPos := nPos + 1;
	aDataOut[nPos] := E_SMPTE_AnalogValue.HIGH; 		nPos := nPos + 1;
	aDataOut[nPos] := E_SMPTE_AnalogValue.LOW; 		nPos := nPos + 1;
	aDataOut[nPos] := E_SMPTE_AnalogValue.HIGH; 		nPos := nPos + 1;
	aDataOut[nPos] := E_SMPTE_AnalogValue.LOW; 		nPos := nPos + 1;
	aDataOut[nPos] := E_SMPTE_AnalogValue.HIGH; 		nPos := nPos + 1;
	
	// 2* 1111
	FOR i:= 0 TO 1 DO 
		aDataOut[nPos] := E_SMPTE_AnalogValue.LOW; 		nPos := nPos + 1;
		aDataOut[nPos] := E_SMPTE_AnalogValue.HIGH; 		nPos := nPos + 1;
		aDataOut[nPos] := E_SMPTE_AnalogValue.LOW; 		nPos := nPos + 1;
		aDataOut[nPos] := E_SMPTE_AnalogValue.HIGH; 		nPos := nPos + 1;
		aDataOut[nPos] := E_SMPTE_AnalogValue.LOW; 		nPos := nPos + 1;
		aDataOut[nPos] := E_SMPTE_AnalogValue.HIGH; 		nPos := nPos + 1;
		aDataOut[nPos] := E_SMPTE_AnalogValue.LOW; 		nPos := nPos + 1;
		aDataOut[nPos] := E_SMPTE_AnalogValue.HIGH; 		nPos := nPos + 1;
	END_FOR
	
	// 1101
	aDataOut[nPos] := E_SMPTE_AnalogValue.LOW; 		nPos := nPos + 1;
	aDataOut[nPos] := E_SMPTE_AnalogValue.HIGH; 		nPos := nPos + 1;
	aDataOut[nPos] := E_SMPTE_AnalogValue.LOW; 		nPos := nPos + 1;
	aDataOut[nPos] := E_SMPTE_AnalogValue.HIGH; 		nPos := nPos + 1;
	aDataOut[nPos] := E_SMPTE_AnalogValue.LOW; 		nPos := nPos + 1;
	aDataOut[nPos] := E_SMPTE_AnalogValue.LOW; 		nPos := nPos + 1;
	aDataOut[nPos] := E_SMPTE_AnalogValue.HIGH; 		nPos := nPos + 1;
	aDataOut[nPos] := E_SMPTE_AnalogValue.LOW; 		nPos := nPos + 1;
ELSE
	// 0011
	aDataOut[nPos] := E_SMPTE_AnalogValue.HIGH; 		nPos := nPos + 1;
	aDataOut[nPos] := E_SMPTE_AnalogValue.HIGH; 		nPos := nPos + 1;
	aDataOut[nPos] := E_SMPTE_AnalogValue.LOW; 		nPos := nPos + 1;
	aDataOut[nPos] := E_SMPTE_AnalogValue.LOW; 		nPos := nPos + 1;
	aDataOut[nPos] := E_SMPTE_AnalogValue.HIGH; 		nPos := nPos + 1;
	aDataOut[nPos] := E_SMPTE_AnalogValue.LOW; 		nPos := nPos + 1;
	aDataOut[nPos] := E_SMPTE_AnalogValue.HIGH; 		nPos := nPos + 1;
	aDataOut[nPos] := E_SMPTE_AnalogValue.LOW; 		nPos := nPos + 1;
	
	// 2* 1111
	FOR i:= 0 TO 1 DO 
		aDataOut[nPos] := E_SMPTE_AnalogValue.HIGH; 		nPos := nPos + 1;
		aDataOut[nPos] := E_SMPTE_AnalogValue.LOW; 		nPos := nPos + 1;
		aDataOut[nPos] := E_SMPTE_AnalogValue.HIGH; 		nPos := nPos + 1;
		aDataOut[nPos] := E_SMPTE_AnalogValue.LOW; 		nPos := nPos + 1;
		aDataOut[nPos] := E_SMPTE_AnalogValue.HIGH; 		nPos := nPos + 1;
		aDataOut[nPos] := E_SMPTE_AnalogValue.LOW; 		nPos := nPos + 1;
		aDataOut[nPos] := E_SMPTE_AnalogValue.HIGH; 		nPos := nPos + 1;
		aDataOut[nPos] := E_SMPTE_AnalogValue.LOW; 		nPos := nPos + 1;
	END_FOR
	
	// 1101
	aDataOut[nPos] := E_SMPTE_AnalogValue.HIGH; 		nPos := nPos + 1;
	aDataOut[nPos] := E_SMPTE_AnalogValue.LOW; 		nPos := nPos + 1;
	aDataOut[nPos] := E_SMPTE_AnalogValue.HIGH; 		nPos := nPos + 1;
	aDataOut[nPos] := E_SMPTE_AnalogValue.LOW; 		nPos := nPos + 1;
	aDataOut[nPos] := E_SMPTE_AnalogValue.HIGH; 		nPos := nPos + 1;
	aDataOut[nPos] := E_SMPTE_AnalogValue.HIGH; 		nPos := nPos + 1;
	aDataOut[nPos] := E_SMPTE_AnalogValue.LOW; 		nPos := nPos + 1;
	aDataOut[nPos] := E_SMPTE_AnalogValue.HIGH; 		nPos := nPos + 1;
END_IF
END_METHOD

END_FUNCTION_BLOCK
